FUNCTION_BLOCK FB_INT_TO_BCD_WORD (* Convert INT to 4 BCD digits *)
  (* Standard: 61499-1; Classification: Simple FB; Function: BCD conversion; Type: INT to WORD *)
  (* Version 0.1, 2008-06-09, JHC, Holobloc Inc, Extended from FBFunction1; deleted QI, QO, STATUS. *)
  (* Version 0.0, 2007-08-27, JHC, Holobloc Inc *)
  (* Compiler header: package fb.rt.math; *)
  (* Compiler classdef: public class FB_INT_TO_BCD_WORD extends FBFunction1 *)
  (* Compiler Java Sun JDK 1.6.0 *)
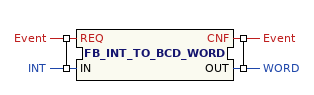
  EVENT_INPUT
    REQ WITH IN; (* Normal Execution Request *)
  END_EVENT
  EVENT_OUTPUT
    CNF WITH OUT; (* Execution Confirmation *)
  END_EVENT
  VAR_INPUT
    IN : INT; (* 0<=IN<=9999 *)
  END_VAR
  VAR_OUTPUT
    OUT : WORD; (* BCD value of IN *)
  END_VAR
END_FUNCTION_BLOCK
